TYPE ES_S1 :
	STRUCT
		Alarm			:ES_ALARM;		
				
		SO2_actVal		:INT;
		SO2_full		:BOOL;
		SO2_fb			:FB_AnalogSensor_full;	

			
	END_STRUCT
END_TYPE

(* stored: Version 1.1.0.1, ProductVersion 3.1.4022.12
   DUT ES_S1: Id {b53ee3b2-7d25-4776-9e12-5ecb9c9d58f2} *)
